// low/high value to controller ---------
      L     DB273.DBD   30; // !!! insert correct AnI !!!
      T     DB276.DBD  218;

      L     DB273.DBD   34; // !!! insert correct AnI !!!
      T     DB276.DBD  222;

NETWORK
TITLE =Sequence organisation

      CLR   ;
      =     M    122.2;

// SFM supply ----------------------------------------------------------------

// analog value to SFM spare -----------------------
      L     DB273.DBD  146;
      T     DB171.DBD 1122; // !!! insert correct SFM !!!

// analog value to SFM spare -----------------------
      L     DB273.DBD  266;
      T     DB171.DBD 1122; // !!! insert correct SFM !!!

// analog value to SFM spare -----------------------
      L     DB273.DBD  386;
      T     DB171.DBD 1122; // !!! insert correct SFM !!!

// sequencer ----------------------------------------------------------------
      A     DB173.DBX   43.1;
      S     DB173.DBX   97.3;

//      CALL  "SeO"          Called in Unit
//       UnitNo:=#UnitNo

NETWORK
TITLE =Auto / Manual

      SET   ;
      AN    M    122.2;
      JC    MODE;
      AN    M    120.1;


// assign PID mode
      S     DB276.DBX  201.4;
      S     DB276.DBX  201.5;


MODE: SET   ;

END_FUNCTION_BLOCK

FUNCTION_BLOCK FB 560
TITLE =
AUTHOR : RR
FAMILY : BOTEC_F1
NAME : OrLiMngA
VERSION : 1.0


VAR_TEMP
  RetVal : WORD ;	//return value
  ValDW : DWORD ;
  ValOK : BOOL ;
  SetValue : DWORD ;
END_VAR
BEGIN
NETWORK
TITLE =Send-/Receive manager telegramtype 1


// Send manager telegramtype 1
      CALL FC   571 (
           RET_VAL                  := #RetVal);

      JBI   OKS1; // Jump, if all OK
// Error evaluation
      L     #RetVal; // Return value
      L     DB33.DBD   84; // Error number from answer
OKS1: NOP   0;

// Receive manager telegramtype 1
      CALL FC   572 (
           RET_VAL                  := #RetVal);

      JBI   OKR1; // Jump, if all OK
// Error evaluation
      L     #RetVal; // Return value
      L     DB33.DBD   84; // Error number from answer
OKR1: NOP   0;


NETWORK
TITLE =Order management

// Telegramtype 1

      CALL FC   560 (
           OrLiDB                   := DB   561,
           RET_VAL                  := #RetVal);

// Telegramtype 2

      CALL FC   560 (
           OrLiDB                   := DB   562,
           RET_VAL                  := #RetVal);

// Telegramtype 3

      CALL FC   560 (
           OrLiDB                   := DB   563,
           RET_VAL                  := #RetVal);

// Telegramtype 4

      CALL FC   560 (
           OrLiDB                   := DB   564,
           RET_VAL                  := #RetVal);

// Telegramtype 5

      CALL FC   560 (
           OrLiDB                   := DB   565,
           RET_VAL                  := #RetVal);


NETWORK
TITLE =Buffer diagnosis

      UC    FB   575;


END_FUNCTION_BLOCK

FUNCTION_BLOCK FB 581
TITLE =
AUTHOR : RR
FAMILY : BOTEC_F1
NAME : CrCA
VERSION : 2.1


VAR_TEMP
  RemotePLCNo : INT ;	//remote PLC number
  RetVal : WORD ;	//return value
END_VAR
BEGIN
NETWORK
TITLE =coupling active bits initialize

      AN    M    101.4;
      JC    NCRC;
      R     DB580.DBX   23.4; // initialize active bits (reset)
      R     DB580.DBX   11.4;
      R     DB580.DBX   47.4;
      R     DB580.DBX   35.4;
      R     DB580.DBX   71.4;
      R     DB580.DBX   59.4;
      R     DB580.DBX   95.4;
      R     DB580.DBX   83.4;
      R     DB580.DBX  119.4;
      R     DB580.DBX  107.4;
      R     DB580.DBX  143.4;
      R     DB580.DBX  131.4;
      R     DB580.DBX  167.4;
      R     DB580.DBX  155.4;
      R     DB580.DBX  191.4;
      R     DB580.DBX  179.4;

NCRC: SET   ;
NETWORK
TITLE =read/write data from/to remote PLC

      NOP   0;

// PLC01
      CALL FB   580 , DB   581 (
           RemotePLCNo              := #RemotePLCNo,
           RetVal                   := #RetVal);

// PLC02
      CALL FB   580 , DB   582 (
           RemotePLCNo              := #RemotePLCNo,
           RetVal                   := #RetVal);

// PLC03
      CALL FB   580 , DB   583 (
           RemotePLCNo              := #RemotePLCNo,
           RetVal                   := #RetVal);

// PLC04
      CALL FB   580 , DB   584 (
           RemotePLCNo              := #RemotePLCNo,
           RetVal                   := #RetVal);

// PLC05
//      CALL  "CCL" , "CCLP05D"
//       RemotePLCNo:=#RemotePLCNo
//       RetVal     :=#RetVal

// PLC06
//      CALL  "CCL" , "CCLP06D"
//       RemotePLCNo:=#RemotePLCNo
//       RetVal     :=#RetVal

// PLC07
//      CALL  "CCL" , "CCLP07D"
//       RemotePLCNo:=#RemotePLCNo
//       RetVal     :=#RetVal

// PLC08
//      CALL  "CCL" , "CCLP08D"
//       RemotePLCNo:=#RemotePLCNo
//       RetVal     :=#RetVal

END_FUNCTION_BLOCK

FUNCTION_BLOCK FB 1000
TITLE =
FAMILY : BOTEC
NAME : UniA
VERSION : 2.0


VAR_TEMP
  UnitNo : INT ;	//unit number
END_VAR
BEGIN
NETWORK
TITLE =general

      L     DB1000.DBW    0;
      T     #UnitNo;

NETWORK
TITLE =analog input's

//      CALL  "AnI"
//       UnitNo:=#UnitNo
//       AnIRec:="U00AnID".AnI1
//       ValPer:=PEW1024

NETWORK
TITLE =PID controller assignment

//      CALL  "PID"
//       UnitNo:=#UnitNo
//       PIDRec:="U00PIDD".PID1
//       SpExt :"U01SeqD".Seq.SFM[x].Sp
//       PVal  :="U00AnID".AnI1.Val
//       OPer  :=PAW1024


//      CALL  "VLT"
//       UnitNo :=#UnitNo
//       VLTRec :="U00VLTD".VLT1
//       BasePEW:=PEW2048
//       COn    :="U00ActD".Act1.Out
//       SpExt  :="U00PIDD".PID1.OVal

NETWORK
TITLE =special input's

//      CALL  "SI1"
//       UnitNo:=#UnitNo
//       SpIRec:="U00SpID".SpI1
//       SpIBit:=E256.0

NETWORK
TITLE =counter

//      CALL  "Cnt"
//       UnitNo:=#UnitNo
//       CntRec:="U00CntD".Cnt1
//       Imp   :="U00SpID".SpI1.Sig
NETWORK
TITLE =message
//
//
// reserved

NETWORK
TITLE =sequence organisation call

      SET   ;
// assignment counter values

//       CALL  "C2S"
//       UnitNo:=#UnitNo
//       CntRec:="U00CntD".Cnt1
//       Enable:="OrgS1"
//       SFMRec:="U00SeqD".Seq.SFM[x]

// assignment analog values

//      L     "U00AnID".AnI1.Val
//      T     "U00SeqD".Seq.SFM[x].Val

      CALL FC    40 (
           UnitNo                   := #UnitNo);

NETWORK
TITLE =mode assignment actuators + PID-controllers

      AN    M    122.2;
      JC    MODE;

      AN    M    120.1;
//      =     "U00ActD".Act1.Auto


MODE: SET   ;
NETWORK
TITLE =actuator's


//      CALL  "Act"
//       UnitNo:=#UnitNo
//       ActRec:="U00ActD".Act1
//       Typ   :=1
//       FBa   :=E0.0
//       FBa2  :=E0.0
//       Out   :=A0.0

END_FUNCTION_BLOCK

FUNCTION_BLOCK FB 1010
TITLE =U001: Wassertank 01
FAMILY : BOTEC_F1
NAME : U001A
VERSION : 2.1


VAR_TEMP
  EStopOK : BOOL ;	//auxiliary flag
  CIP : BOOL ;	//CIP Program Selected
  xTmp : BOOL ;	//Temporary Bool(free for general use)
  DummyBool : BOOL ;	//Temporary Bool(free for general use)
  UnitNo : INT ;	//unit number
  UnitFB : INT ;	//unit expansion FB number
  rTmp : REAL ;	//Temporary REAL (free for general use)
  iTmp : INT ;	//Temporary INT (free for general use)
  DummyInt : INT ;	//Temporary INT (free for general use)
  dTmp : DINT ;	//Temporary DINT (free for general use)
END_VAR
BEGIN
NETWORK
TITLE =general

      CLR   ;
      =     #xTmp;
      =     #EStopOK;

      L     DB1010.DBW    0;
      T     #UnitNo;
      L     DB1010.DBW    2;
      T     #UnitFB;

NETWORK
TITLE =analog inputs

      NOP   0;
// LI_T1 AnI 001 Inhalt Tank 1
      CALL FC    24 (
           UnitNo                   := #UnitNo,
           AnIRec                   := DB2013.LI_T1,
           ValPer                   := DB302.DBW   64);

NETWORK
TITLE =Universal value

      NOP   0;
// unv001 UnV 001 Process Status
      CALL FC    27 (
           UnitNo                   := #UnitNo,
           UnVRec                   := DB2015.unv001,
           ValExt                   := DB2015.DBD  234);

// unv002 UnV 002 Universal Value 02
      CALL FC    27 (
           UnitNo                   := #UnitNo,
           UnVRec                   := DB2015.unv002,
           ValExt                   := DB2015.DBD  362);

// unv003 UnV 003 Universal Value 03
      CALL FC    27 (
           UnitNo                   := #UnitNo,
           UnVRec                   := DB2015.unv003,
           ValExt                   := DB2015.DBD  490);

NETWORK
TITLE =special inputs

      NOP   0;
// LS_LLL_T1 SpI 001
      CALL FC    14 (
           UnitNo                   := #UnitNo,
           SpIRec                   := DB2011.LS_LLL_T1,
           SpIBit                   := I     70.0);

// LS_HL_T1 SpI 002
      CALL FC    14 (
           UnitNo                   := #UnitNo,
           SpIRec                   := DB2011.LS_HL_T1,
           SpIBit                   := I     69.5);

// RM_NI_T1_VV SpI 004 Vacuumventil Tank 1
      CALL FC    14 (
           UnitNo                   := #UnitNo,
           SpIRec                   := DB2011.RM_NI_T1_VV,
           SpIBit                   := I    186.5);

// LS_LL_T1 SpI 005 (als Leermeldung ausgelegt)
      CALL FC    14 (
           UnitNo                   := #UnitNo,
           SpIRec                   := DB2011.LS_LL_T1,
           SpIBit                   := I     69.6);

// RM_NI_T1_K4_AUF SpI 006 Klappe vor Filter Tank 1
      CALL FC    14 (
           UnitNo                   := #UnitNo,
           SpIRec                   := DB2011.RM_NI_T1_K4_AUF,
           SpIBit                   := I    186.3);

// RM_NI_T1_K4_ZU SpI 007 Klappe vor Filter Tank 1
      CALL FC    14 (
           UnitNo                   := #UnitNo,
           SpIRec                   := DB2011.RM_NI_T1_K4_ZU,
           SpIBit                   := I    186.4);

// RM_NI_T1_K2 SpI 008 Handklappe Tank 1
      CALL FC    14 (
           UnitNo                   := #UnitNo,
           SpIRec                   := DB2011.RM_NI_T1_K2,
           SpIBit                   := I     71.1);

// RM_NI_T1_K3 SpI 010 Handklappe Tank 1
      CALL FC    14 (
           UnitNo                   := #UnitNo,
           SpIRec                   := DB2011.RM_NI_T1_K3,
           SpIBit                   := I     71.2);

// LABOR_FREIG_T1 SpI 011 SCHLUESSELSCHALTER LABOR
      CALL FC    14 (
           UnitNo                   := #UnitNo,
           SpIRec                   := DB2011.LABOR_FREIG_T1,
           SpIBit                   := I    258.0);

NETWORK
TITLE =messages

      NOP   0;
// msg001 Msg 001 Message 01
      CALL FC    16 (
           UnitNo                   := #UnitNo,
           MsgRec                   := DB2017.msg001,
           MsgBit                   := DB2017.DBX   82.7);

// msg002 Msg 002 Message 02
      CALL FC    16 (
           UnitNo                   := #UnitNo,
           MsgRec                   := DB2017.msg002,
           MsgBit                   := DB2017.DBX  142.7);

NETWORK
TITLE =unit supply

      UC    FB [#UnitFB];

NETWORK
TITLE =T1_A10
// Act 005
// Box           : Ventilinsel 2
// Input address : I317.0
// Output address: Q317.0
      CALL FC    70 (
           UnitNo                   := #UnitNo,
           ActRec                   := DB2010.T1_A10,
           Typ                      := 1,
           FBa                      := #xTmp,
           FBa2                     := I    317.0,
           Out                      := Q    317.0);

NETWORK
TITLE =T1_A9
// Act 006
// Box           : Ventilinsel 2
// Input address : I319.0
// Output address: Q319.0
      CALL FC    70 (
           UnitNo                   := #UnitNo,
           ActRec                   := DB2010.T1_A9,
           Typ                      := 1,
           FBa                      := #xTmp,
           FBa2                     := I    319.0,
           Out                      := Q    319.0);

NETWORK
TITLE =T1_A12
// Act 007
// Box           : Ventilinsel 2
// Input address : I321.0
// Output address: Q321.0
      CALL FC    70 (
           UnitNo                   := #UnitNo,
           ActRec                   := DB2010.T1_A12,
           Typ                      := 1,
           FBa                      := #xTmp,
           FBa2                     := I    321.0,
           Out                      := Q    321.0);

NETWORK
TITLE =T1_A7
// Act 008
// Box           : Ventilinsel 2
// Input address : I323.0
// Output address: Q323.0
      CALL FC    70 (
           UnitNo                   := #UnitNo,
           ActRec                   := DB2010.T1_A7,
           Typ                      := 1,
           FBa                      := #xTmp,
           FBa2                     := I    323.0,
           Out                      := Q    323.0);

NETWORK
TITLE =T1_A8
// Act 009
// Box           : Ventilinsel 3
// Input address : I325.0
// Output address: Q325.0
      CALL FC    70 (
           UnitNo                   := #UnitNo,
           ActRec                   := DB2010.T1_A8,
           Typ                      := 1,
           FBa                      := #xTmp,
           FBa2                     := I    325.0,
           Out                      := Q    325.0);

NETWORK
TITLE =T1_A5
// Act 010
// Box           : Ventilinsel 3
// Input address : I327.0
// Output address: Q327.0
      CALL FC    70 (
           UnitNo                   := #UnitNo,
           ActRec                   := DB2010.T1_A5,
           Typ                      := 1,
           FBa                      := #xTmp,
           FBa2                     := I    327.0,
           Out                      := Q    327.0);

NETWORK
TITLE =T1_A11
// Act 011
// Box           : Ventilinsel 3
// Input address : I329.0
// Output address: Q329.0
      CALL FC    70 (
           UnitNo                   := #UnitNo,
           ActRec                   := DB2010.T1_A11,
           Typ                      := 1,
           FBa                      := #xTmp,
           FBa2                     := I    329.0,
           Out                      := Q    329.0);

NETWORK
TITLE =T1_A14
// Act 012
// Box           : Ventilinsel 4
// Input address : I331.0
// Output address: Q331.0
      CALL FC    70 (
           UnitNo                   := #UnitNo,
           ActRec                   := DB2010.T1_A14,
           Typ                      := 1,
           FBa                      := #xTmp,
           FBa2                     := I    331.0,
           Out                      := Q    331.0);

NETWORK
TITLE =T1_A15
// Act 013
// Box           : Ventilinsel 4
// Input address : I333.0
// Output address: Q333.0
      CALL FC    70 (
           UnitNo                   := #UnitNo,
           ActRec                   := DB2010.T1_A15,
           Typ                      := 0,
           FBa                      := #xTmp,
           FBa2                     := I    333.0,
           Out                      := Q    333.0);

NETWORK
TITLE =T1_RR1
// Act 014
// Box           : Ventilinsel 4
// Input address : I335.0
// Output address: Q335.0
      CALL FC    70 (
           UnitNo                   := #UnitNo,
           ActRec                   := DB2010.T1_RR1,
           Typ                      := 1,
           FBa                      := #xTmp,
           FBa2                     := I    335.0,
           Out                      := Q    335.0);

NETWORK
TITLE =RV1_T1  RV1_T1
// Act 015
// Box           : VS1-BB
// Input address : I296.0
// Output address: Q296.0
      CALL FC    70 (
           UnitNo                   := #UnitNo,
           ActRec                   := DB2010.RV1_T1,
           Typ                      := 1,
           FBa                      := #xTmp,
           FBa2                     := I    296.0,
           Out                      := Q    296.0);

NETWORK
TITLE =B6F_T1  B6F_T1
// Act 016
// Box           : VS1-BB
// Input address : I296.4
// Output address: Q296.4
      CALL FC    70 (
           UnitNo                   := #UnitNo,
           ActRec                   := DB2010.B6F_T1,
           Typ                      := 1,
           FBa                      := #xTmp,
           FBa2                     := I    296.4,
           Out                      := Q    296.4);

NETWORK
TITLE =H6F_T1  H6F_T1
// Act 017
// Box           : VS1-BB
// Input address : I296.3
// Output address: Q296.3
      CALL FC    70 (
           UnitNo                   := #UnitNo,
           ActRec                   := DB2010.H6F_T1,
           Typ                      := 1,
           FBa                      := #xTmp,
           FBa2                     := I    296.3,
           Out                      := Q    296.3);

NETWORK
TITLE =J6F_T1  J6F_T1
// Act 018
// Box           : VS1-BB
// Input address : I296.5
// Output address: Q296.5
      CALL FC    70 (
           UnitNo                   := #UnitNo,
           ActRec                   := DB2010.J6F_T1,
           Typ                      := 1,
           FBa                      := #xTmp,
           FBa2                     := I    296.5,
           Out                      := Q    296.5);

NETWORK
TITLE =L6F_T1  L6F_T1
// Act 019
// Box           : VS1-BB
// Input address : I296.6
// Output address: Q296.6
      CALL FC    70 (
           UnitNo                   := #UnitNo,
           ActRec                   := DB2010.L6F_T1,
           Typ                      := 1,
           FBa                      := #xTmp,
           FBa2                     := I    296.6,
           Out                      := Q    296.6);

NETWORK
TITLE =D6_T1  D6_T1
// Act 020
// Box           : VS1-BB
// Input address : I297.0
// Output address: Q297.0
      CALL FC    70 (
           UnitNo                   := #UnitNo,
           ActRec                   := DB2010.D6_T1,
           Typ                      := 1,
           FBa                      := #xTmp,
           FBa2                     := I    297.0,
           Out                      := Q    297.0);

NETWORK
TITLE =B6_T1  B6_T1
// Act 021
// Box           : VS1-BB
// Input address : I296.7
// Output address: Q296.7
      CALL FC    70 (
           UnitNo                   := #UnitNo,
           ActRec                   := DB2010.B6_T1,
           Typ                      := 1,
           FBa                      := #xTmp,
           FBa2                     := I    296.7,
           Out                      := Q    296.7);

NETWORK
TITLE =A_T1  A_T1
// Act 022
// Box           : VS1-BB
// Input address : I296.1
// Output address: Q296.1
      CALL FC    70 (
           UnitNo                   := #UnitNo,
           ActRec                   := DB2010.A_T1,
           Typ                      := 1,
           FBa                      := #xTmp,
           FBa2                     := I    296.1,
           Out                      := Q    296.1);

NETWORK
TITLE =B_T1  B_T1
// Act 023
// Box           : VS1-BB
// Input address : I296.2
// Output address: Q296.2
      CALL FC    70 (
           UnitNo                   := #UnitNo,
           ActRec                   := DB2010.B_T1,
           Typ                      := 1,
           FBa                      := #xTmp,
           FBa2                     := I    296.2,
           Out                      := Q    296.2);

NETWORK
TITLE =CF_T1
// Act 024
// Box           : Ventilinsel 1
// Input address : I16.1
// Output address: Q16.1
      CALL FC    70 (
           UnitNo                   := #UnitNo,
           ActRec                   := DB2010.CF_T1,
           Typ                      := 1,
           FBa                      := #xTmp,
           FBa2                     := I     16.1,
           Out                      := Q     16.1);

NETWORK
TITLE =RW5_T1  Ansteuerung Befüllventil
// Act 026
// Box           : Ventilinsel 1
// Input address : I16.0
// Output address: Q16.0
      CALL FC    70 (
           UnitNo                   := #UnitNo,
           ActRec                   := DB2010.RW5_T1,
           Typ                      := 1,
           FBa                      := #xTmp,
           FBa2                     := I     16.0,
           Out                      := Q     16.0);

NETWORK
TITLE =RW6_T1  RW6_T1
// Act 027
// Box           : VS1-BB
// Input address : I297.1
// Output address: Q297.1
      CALL FC    70 (
           UnitNo                   := #UnitNo,
           ActRec                   := DB2010.RW6_T1,
           Typ                      := 1,
           FBa                      := #xTmp,
           FBa2                     := I    297.1,
           Out                      := Q    297.1);

NETWORK
TITLE =VR_T1  VR_T1
// Act 029
// Box           : VS1-BB
// Output address: Q297.2
      CALL FC    70 (
           UnitNo                   := #UnitNo,
           ActRec                   := DB2010.VR_T1,
           Typ                      := 0,
           FBa                      := #xTmp,
           FBa2                     := #xTmp,
           Out                      := Q    297.2);

NETWORK
TITLE =T1_V3
// Act 030
// Box           : Ventilinsel 5
// Input address : I340.2
// Output address: Q340.2
//      CALL  "Act"
//       UnitNo:=#UnitNo
//       ActRec:="U001ActD".T1_V3
//       Typ   :=0
//       FBa   :=#xTmp
//       FBa2  :="T1_V3GSC"
//       Out   :="T1_V3O"

NETWORK
TITLE =ML_LABORFREIGABE_T1
// Act 031
// Box           : LT-CIP
// Output address: Q258.0
      CALL FC    70 (
           UnitNo                   := #UnitNo,
           ActRec                   := DB2010.ML_LABORFREIGABE_T1,
           Typ                      := 0,
           FBa                      := #xTmp,
           FBa2                     := #xTmp,
           Out                      := Q    258.0);

END_FUNCTION_BLOCK

FUNCTION_BLOCK FB 1011
TITLE =U001: Water Tank 1
FAMILY : BOTEC_F1
NAME : UniE
VERSION : 1.2


VAR_TEMP
  CIP : BOOL ;	//CIP active
  UNIM : BOOL ;	//Unit Not In Maintenance
  GenRel : BOOL ;	//general OK (emergency and maintenance OK)
  EStopOK : BOOL ;	//emergency OK
  UnitNo : INT ;	//unit number
  xTmp : BOOL ;	//Temporary Bool
  iTmp : INT ;	//Temporary INT
  rTmp : REAL ;	//Temporary REAL
  dTmp : DINT ;	//Temporary DINT (free for general use)
  RetValInt : INT ;	//return value
END_VAR
BEGIN
NETWORK
TITLE =General

      SET   ;
// Simulation ---------------------------------------------------------------
      A     DB1011.DBX 1357.7;
      CC    FB  1019; // "U001Sim"
      A     DB1011.DBX   17.3;
      =     DB1011.DBX 1357.7; //Help bit for simulation

// get unit number ----------------------------------------------------------
      L     DB1010.DBW    0;
      T     #UnitNo;

// communication ------------------------------------------------------------
      UC    FB  1015; // U001Com

NETWORK
TITLE =Sequence organisation

      CLR   ;
      =     M    122.2;

// CIP Counter
      CALL FC    29 (
           UnitNo                   := #UnitNo,
           Value                    := DB1015.DBD   54,
           Enable                   := TRUE,
           Down                     := FALSE,
           OriginDetect             := 0.000000e+000,
           MaxDiffPS                := 1.000000e+000,
           SFMRec                   := DB1011.Seq.SFM[15],
           ValueOld                 := DB1011.DBD 1418);

// sequencer ----------------------------------------------------------------
      A     DB1013.DBX   43.1;
      S     DB1013.DBX   97.3;

      CALL FC    40 (
           UnitNo                   := #UnitNo);

END_FUNCTION_BLOCK

FUNCTION_BLOCK FB 1020
TITLE =U002: Wassertank 02
FAMILY : BOTEC_F1
NAME : U002A
VERSION : 2.1


VAR_TEMP
  EStopOK : BOOL ;	//auxiliary flag
  CIP : BOOL ;	//CIP Program Selected
  xTmp : BOOL ;	//Temporary Bool(free for general use)
  DummyBool : BOOL ;	//Temporary Bool(free for general use)
  UnitNo : INT ;	//unit number
  UnitFB : INT ;	//unit expansion FB number
  rTmp : REAL ;	//Temporary REAL (free for general use)
  iTmp : INT ;	//Temporary INT (free for general use)
  DummyInt : INT ;	//Temporary INT (free for general use)
  dTmp : DINT ;	//Temporary DINT (free for general use)
END_VAR
BEGIN
NETWORK
TITLE =general

      CLR   ;
      =     #xTmp;
      =     #EStopOK;

      L     DB1020.DBW    0;
      T     #UnitNo;
      L     DB1020.DBW    2;
      T     #UnitFB;

NETWORK
TITLE =analog inputs

      NOP   0;
// LI_T2 AnI 001 Inhalt Tank 2
      CALL FC    24 (
           UnitNo                   := #UnitNo,
           AnIRec                   := DB2023.LI_T2,
           ValPer                   := DB302.DBW   66);

NETWORK
TITLE =Universal value

      NOP   0;
// unv001 UnV 001 Process Status
      CALL FC    27 (
           UnitNo                   := #UnitNo,
           UnVRec                   := DB2025.unv001,
           ValExt                   := DB2025.DBD  234);

// unv002 UnV 002 Universal Value 02
      CALL FC    27 (
           UnitNo                   := #UnitNo,
           UnVRec                   := DB2025.unv002,
           ValExt                   := DB2025.DBD  362);

// unv003 UnV 003 Universal Value 03
      CALL FC    27 (
           UnitNo                   := #UnitNo,
           UnVRec                   := DB2025.unv003,
           ValExt                   := DB2025.DBD  490);

NETWORK
TITLE =special inputs

      NOP   0;
// LS_LLL_T2 SpI 001
      CALL FC    14 (
           UnitNo                   := #UnitNo,
           SpIRec                   := DB2021.LS_LLL_T2,
           SpIBit                   := I     71.7);

// LS_HL_T2 SpI 002
      CALL FC    14 (
           UnitNo                   := #UnitNo,
           SpIRec                   := DB2021.LS_HL_T2,
           SpIBit                   := I     69.7);

// LS_LL_T2 SpI 005
      CALL FC    14 (
           UnitNo                   := #UnitNo,
           SpIRec                   := DB2021.LS_LL_T2,
           SpIBit                   := I     70.1);

// RM_NI_T2_K2 SpI 008
      CALL FC    14 (
           UnitNo                   := #UnitNo,
           SpIRec                   := DB2021.RM_NI_T2_K2,
           SpIBit                   := I     61.6);

// RM_NI_T2_K3 SpI 010
      CALL FC    14 (
           UnitNo                   := #UnitNo,
           SpIRec                   := DB2021.RM_NI_T2_K3,
           SpIBit                   := I     61.7);

// LABOR_FREIG_T2 SpI 011 SCHLUESSELSCHALTER LABOR
      CALL FC    14 (
           UnitNo                   := #UnitNo,
           SpIRec                   := DB2021.LABOR_FREIG_T2,
           SpIBit                   := I    258.1);

NETWORK
TITLE =messages

      NOP   0;
// msg001 Msg 001 Message 01
      CALL FC    16 (
           UnitNo                   := #UnitNo,
           MsgRec                   := DB2027.msg001,
           MsgBit                   := DB2027.DBX   82.7);

// msg002 Msg 002 Message 02
      CALL FC    16 (
           UnitNo                   := #UnitNo,
           MsgRec                   := DB2027.msg002,
           MsgBit                   := DB2027.DBX  142.7);

NETWORK
TITLE =unit supply

      UC    FB [#UnitFB];

NETWORK
TITLE =T2_A10
// Act 005
// Box           : Ventilinsel 2
// Input address : I316.7
// Output address: Q316.7
      CALL FC    70 (
           UnitNo                   := #UnitNo,
           ActRec                   := DB2020.T2_A10,
           Typ                      := 1,
           FBa                      := #xTmp,
           FBa2                     := I    316.7,
           Out                      := Q    316.7);

NETWORK
TITLE =T2_A9
// Act 006
// Box           : Ventilinsel 2
// Input address : I318.7
// Output address: Q318.7
      CALL FC    70 (
           UnitNo                   := #UnitNo,
           ActRec                   := DB2020.T2_A9,
           Typ                      := 1,
           FBa                      := #xTmp,
           FBa2                     := I    318.7,
           Out                      := Q    318.7);

NETWORK
TITLE =T2_A12
// Act 007
// Box           : Ventilinsel 2
// Input address : I320.7
// Output address: Q320.7
      CALL FC    70 (
           UnitNo                   := #UnitNo,
           ActRec                   := DB2020.T2_A12,
           Typ                      := 1,
           FBa                      := #xTmp,
           FBa2                     := I    320.7,
           Out                      := Q    320.7);

NETWORK
TITLE =T2_A7
// Act 008
// Box           : Ventilinsel 2
// Input address : I322.7
// Output address: Q322.7
      CALL FC    70 (
           UnitNo                   := #UnitNo,
           ActRec                   := DB2020.T2_A7,
           Typ                      := 1,
           FBa                      := #xTmp,
           FBa2                     := I    322.7,
           Out                      := Q    322.7);

NETWORK
TITLE =T2_A8
// Act 009
// Box           : Ventilinsel 3
// Input address : I324.7
// Output address: Q324.7
      CALL FC    70 (
           UnitNo                   := #UnitNo,
           ActRec                   := DB2020.T2_A8,
           Typ                      := 1,
           FBa                      := #xTmp,
           FBa2                     := I    324.7,
           Out                      := Q    324.7);

NETWORK
TITLE =T2_A5
// Act 010
// Box           : Ventilinsel 3
// Input address : I326.7
// Output address: Q326.7
      CALL FC    70 (
           UnitNo                   := #UnitNo,
           ActRec                   := DB2020.T2_A5,
           Typ                      := 1,
           FBa                      := #xTmp,
           FBa2                     := I    326.7,
           Out                      := Q    326.7);

NETWORK
TITLE =T2_A11
// Act 011
// Box           : Ventilinsel 3
// Input address : I328.7
// Output address: Q328.7
      CALL FC    70 (
           UnitNo                   := #UnitNo,
           ActRec                   := DB2020.T2_A11,
           Typ                      := 1,
           FBa                      := #xTmp,
           FBa2                     := I    328.7,
           Out                      := Q    328.7);

NETWORK
TITLE =T2_A14
// Act 012
// Box           : Ventilinsel 4
// Input address : I330.7
// Output address: Q330.7
      CALL FC    70 (
           UnitNo                   := #UnitNo,
           ActRec                   := DB2020.T2_A14,
           Typ                      := 1,
           FBa                      := #xTmp,
           FBa2                     := I    330.7,
           Out                      := Q    330.7);

NETWORK
TITLE =T2_A15
// Act 013
// Box           : Ventilinsel 4
// Input address : I332.7
// Output address: Q332.7
      CALL FC    70 (
           UnitNo                   := #UnitNo,
           ActRec                   := DB2020.T2_A15,
           Typ                      := 0,
           FBa                      := #xTmp,
           FBa2                     := I    332.7,
           Out                      := Q    332.7);

NETWORK
TITLE =T2_RR1
// Act 014
// Box           : Ventilinsel 4
// Input address : I334.7
// Output address: Q334.7
      CALL FC    70 (
           UnitNo                   := #UnitNo,
           ActRec                   := DB2020.T2_RR1,
           Typ                      := 1,
           FBa                      := #xTmp,
           FBa2                     := I    334.7,
           Out                      := Q    334.7);

NETWORK
TITLE =RV1_T2  RV1_T2
// Act 015
// Box           : VS1-BB
// Input address : I297.3
// Output address: Q297.3
      CALL FC    70 (
           UnitNo                   := #UnitNo,
           ActRec                   := DB2020.RV1_T2,
           Typ                      := 1,
           FBa                      := #xTmp,
           FBa2                     := I    297.3,
           Out                      := Q    297.3);

NETWORK
TITLE =B6F_T2  B6F_T2
// Act 016
// Box           : VS1-BB
// Input address : I297.7
// Output address: Q297.7
      CALL FC    70 (
           UnitNo                   := #UnitNo,
           ActRec                   := DB2020.B6F_T2,
           Typ                      := 1,
           FBa                      := #xTmp,
           FBa2                     := I    297.7,
           Out                      := Q    297.7);

NETWORK
TITLE =H6F_T2  H6F_T2
// Act 017
// Box           : VS1-BB
// Input address : I297.6
// Output address: Q297.6
      CALL FC    70 (
           UnitNo                   := #UnitNo,
           ActRec                   := DB2020.H6F_T2,
           Typ                      := 1,
           FBa                      := #xTmp,
           FBa2                     := I    297.6,
           Out                      := Q    297.6);

NETWORK
TITLE =J6F_T2  J6F_T2
// Act 018
// Box           : VS1-BB
// Input address : I298.0
// Output address: Q298.0
      CALL FC    70 (
           UnitNo                   := #UnitNo,
           ActRec                   := DB2020.J6F_T2,
           Typ                      := 1,
           FBa                      := #xTmp,
           FBa2                     := I    298.0,
           Out                      := Q    298.0);

NETWORK
TITLE =L6F_T2  L6F_T2
// Act 019
// Box           : VS1-BB
// Input address : I298.1
// Output address: Q298.1
      CALL FC    70 (
           UnitNo                   := #UnitNo,
           ActRec                   := DB2020.L6F_T2,
           Typ                      := 1,
           FBa                      := #xTmp,
           FBa2                     := I    298.1,
           Out                      := Q    298.1);

NETWORK
TITLE =D6_T2  D6_T2
// Act 020
// Box           : VS1-BB
// Input address : I298.3
// Output address: Q298.3
      CALL FC    70 (
           UnitNo                   := #UnitNo,
           ActRec                   := DB2020.D6_T2,
           Typ                      := 1,
           FBa                      := #xTmp,
           FBa2                     := I    298.3,
           Out                      := Q    298.3);

NETWORK
TITLE =B6_T2  B6_T2
// Act 021
// Box           : VS1-BB
// Input address : I298.2
// Output address: Q298.2
      CALL FC    70 (
           UnitNo                   := #UnitNo,
           ActRec                   := DB2020.B6_T2,
           Typ                      := 1,
           FBa                      := #xTmp,
           FBa2                     := I    298.2,
           Out                      := Q    298.2);

NETWORK
TITLE =A_T2  A_T2
// Act 022
// Box           : VS1-BB
// Input address : I297.4
// Output address: Q297.4
      CALL FC    70 (
           UnitNo                   := #UnitNo,
           ActRec                   := DB2020.A_T2,
           Typ                      := 1,
           FBa                      := #xTmp,
           FBa2                     := I    297.4,
           Out                      := Q    297.4);

NETWORK
TITLE =B_T2  B_T2
// Act 023
// Box           : VS1-BB
// Input address : I297.5
// Output address: Q297.5
      CALL FC    70 (
           UnitNo                   := #UnitNo,
           ActRec                   := DB2020.B_T2,
           Typ                      := 1,
           FBa                      := #xTmp,
           FBa2                     := I    297.5,
           Out                      := Q    297.5);

NETWORK
TITLE =CF_T2
// Act 024
// Box           : Ventilinsel 1
// Input address : I16.2
// Output address: Q16.2
      CALL FC    70 (
           UnitNo                   := #UnitNo,
           ActRec                   := DB2020.CF_T2,
           Typ                      := 1,
           FBa                      := #xTmp,
           FBa2                     := I     16.2,
           Out                      := Q     16.2);

NETWORK
TITLE =VR_T2  VR_T2
// Act 029
// Box           : VS1-BB
// Output address: Q298.4
      CALL FC    70 (
           UnitNo                   := #UnitNo,
           ActRec                   := DB2020.VR_T2,
           Typ                      := 0,
           FBa                      := #xTmp,
           FBa2                     := #xTmp,
           Out                      := Q    298.4);

NETWORK
TITLE =ML_LABORFREIGABE_T2
// Act 031
// Box           : LT-CIP
// Output address: Q258.1
      CALL FC    70 (
           UnitNo                   := #UnitNo,
           ActRec                   := DB2020.ML_LABORFREIGABE_T2,
           Typ                      := 0,
           FBa                      := #xTmp,
           FBa2                     := #xTmp,
           Out                      := Q    258.1);

END_FUNCTION_BLOCK

FUNCTION_BLOCK FB 1021
TITLE =U002: Water Tank 2
FAMILY : BOTEC_F1
NAME : UniE
VERSION : 1.2


VAR_TEMP
  CIP : BOOL ;	//CIP active
  UNIM : BOOL ;	//Unit Not In Maintenance
  GenRel : BOOL ;	//general OK (emergency and maintenance OK)
  EStopOK : BOOL ;	//emergency OK
  UnitNo : INT ;	//unit number
  xTmp : BOOL ;	//Temporary Bool
  iTmp : INT ;	//Temporary INT
  rTmp : REAL ;	//Temporary REAL
  dTmp : DINT ;	//Temporary DINT (free for general use)
  RetValInt : INT ;	//return value
END_VAR
BEGIN
NETWORK
TITLE =General

      SET   ;
// Simulation ---------------------------------------------------------------
      A     DB1021.DBX 1357.7;
      CC    FB  1029; // "WT02Sim"
      A     DB1021.DBX   17.3;
      =     DB1021.DBX 1357.7; //Help bit for simulation

// get unit number ----------------------------------------------------------
      L     DB1020.DBW    0;
      T     #UnitNo;


// communication ------------------------------------------------------------
      UC    FB  1025; // WT02Com

NETWORK
TITLE =Sequence organisation

      CLR   ;
      =     M    122.2;

// CIP Counter
      CALL FC    29 (
           UnitNo                   := #UnitNo,
           Value                    := DB1025.DBD   54,
           Enable                   := TRUE,
           Down                     := FALSE,
           OriginDetect             := 0.000000e+000,
           MaxDiffPS                := 1.000000e+000,
           SFMRec                   := DB1021.Seq.SFM[15],
           ValueOld                 := DB1021.DBD 1418);

// sequencer ----------------------------------------------------------------
      A     DB1023.DBX   43.1;
      S     DB1023.DBX   97.3;

      CALL FC    40 (
           UnitNo                   := #UnitNo);

END_FUNCTION_BLOCK

FUNCTION_BLOCK FB 1030
TITLE =U003: Wassertank 03
FAMILY : BOTEC_F1
NAME : U003A
VERSION : 2.1


VAR_TEMP
  EStopOK : BOOL ;	//auxiliary flag
  CIP : BOOL ;	//CIP Program Selected
  xTmp : BOOL ;	//Temporary Bool(free for general use)
  DummyBool : BOOL ;	//Temporary Bool(free for general use)
  UnitNo : INT ;	//unit number
  UnitFB : INT ;	//unit expansion FB number
  rTmp : REAL ;	//Temporary REAL (free for general use)
  iTmp : INT ;	//Temporary INT (free for general use)
  DummyInt : INT ;	//Temporary INT (free for general use)
  dTmp : DINT ;	//Temporary DINT (free for general use)
END_VAR
BEGIN
NETWORK
TITLE =general

      CLR   ;
      =     #xTmp;
      =     #EStopOK;

      L     DB1030.DBW    0;
      T     #UnitNo;
      L     DB1030.DBW    2;
      T     #UnitFB;

NETWORK
TITLE =analog inputs

      NOP   0;
// LI_T3 AnI 001 Inhalt Tank 3
      CALL FC    24 (
           UnitNo                   := #UnitNo,
           AnIRec                   := DB2033.LI_T3,
           ValPer                   := DB302.DBW   68);

NETWORK
TITLE =Universal value

      NOP   0;
// unv001 UnV 001 Process Status
      CALL FC    27 (
           UnitNo                   := #UnitNo,
           UnVRec                   := DB2035.unv001,
           ValExt                   := DB2035.DBD  234);

// unv002 UnV 002 Universal Value 02
      CALL FC    27 (
           UnitNo                   := #UnitNo,
           UnVRec                   := DB2035.unv002,
           ValExt                   := DB2035.DBD  362);

// unv003 UnV 003 Universal Value 03
      CALL FC    27 (
           UnitNo                   := #UnitNo,
           UnVRec                   := DB2035.unv003,
           ValExt                   := DB2035.DBD  490);

NETWORK
TITLE =special inputs

      NOP   0;
// LS_LLL_T3 SpI 001
      CALL FC    14 (
           UnitNo                   := #UnitNo,
           SpIRec                   := DB2031.LS_LLL_T3,
           SpIBit                   := I     60.1);

// LS_HL_T3 SpI 002
      CALL FC    14 (
           UnitNo                   := #UnitNo,
           SpIRec                   := DB2031.LS_HL_T3,
           SpIBit                   := I     70.2);

// LS_LL_T3 SpI 005
      CALL FC    14 (
           UnitNo                   := #UnitNo,
           SpIRec                   := DB2031.LS_LL_T3,
           SpIBit                   := I     60.0);

// RM_NI_T3_K2 SpI 008
      CALL FC    14 (
           UnitNo                   := #UnitNo,
           SpIRec                   := DB2031.RM_NI_T3_K2,
           SpIBit                   := I     60.6);

// RM_NI_T3_K3 SpI 010
      CALL FC    14 (
           UnitNo                   := #UnitNo,
           SpIRec                   := DB2031.RM_NI_T3_K3,
           SpIBit                   := I     69.0);

// LABOR_FREIG_T3 SpI 011 SCHLUESSELSCHALTER LABOR
      CALL FC    14 (
           UnitNo                   := #UnitNo,
           SpIRec                   := DB2031.LABOR_FREIG_T3,
           SpIBit                   := I    258.2);

NETWORK
TITLE =messages

      NOP   0;
// msg001 Msg 001 Message 01
      CALL FC    16 (
           UnitNo                   := #UnitNo,
           MsgRec                   := DB2037.msg001,
           MsgBit                   := DB2037.DBX   82.7);

// msg002 Msg 002 Message 02
      CALL FC    16 (
           UnitNo                   := #UnitNo,
           MsgRec                   := DB2037.msg002,
           MsgBit                   := DB2037.DBX  142.7);

NETWORK
TITLE =unit supply

      UC    FB [#UnitFB];

NETWORK
TITLE =T3_A10
// Act 005
// Box           : Ventilinsel 2
// Input address : I316.6
// Output address: Q316.6
      CALL FC    70 (
           UnitNo                   := #UnitNo,
           ActRec                   := DB2030.T3_A10,
           Typ                      := 1,
           FBa                      := #xTmp,
           FBa2                     := I    316.6,
           Out                      := Q    316.6);

NETWORK
TITLE =T3_A9
// Act 006
// Box           : Ventilinsel 2
// Input address : I318.6
// Output address: Q318.6
      CALL FC    70 (
           UnitNo                   := #UnitNo,
           ActRec                   := DB2030.T3_A9,
           Typ                      := 1,
           FBa                      := #xTmp,
           FBa2                     := I    318.6,
           Out                      := Q    318.6);

NETWORK
TITLE =T3_A12
// Act 007
// Box           : Ventilinsel 2
// Input address : I320.6
// Output address: Q320.6
      CALL FC    70 (
           UnitNo                   := #UnitNo,
           ActRec                   := DB2030.T3_A12,
           Typ                      := 1,
           FBa                      := #xTmp,
           FBa2                     := I    320.6,
           Out                      := Q    320.6);

NETWORK
TITLE =T3_A7
// Act 008
// Box           : Ventilinsel 2
// Input address : I322.6
// Output address: Q322.6
      CALL FC    70 (
           UnitNo                   := #UnitNo,
           ActRec                   := DB2030.T3_A7,
           Typ                      := 1,
           FBa                      := #xTmp,
           FBa2                     := I    322.6,
           Out                      := Q    322.6);

NETWORK
TITLE =T3_A8
// Act 009
// Box           : Ventilinsel 3
// Input address : I324.6
// Output address: Q324.6
      CALL FC    70 (
           UnitNo                   := #UnitNo,
           ActRec                   := DB2030.T3_A8,
           Typ                      := 1,
           FBa                      := #xTmp,
           FBa2                     := I    324.6,
           Out                      := Q    324.6);

NETWORK
TITLE =T3_A5
// Act 010
// Box           : Ventilinsel 3
// Input address : I326.6
// Output address: Q326.6
      CALL FC    70 (
           UnitNo                   := #UnitNo,
           ActRec                   := DB2030.T3_A5,
           Typ                      := 1,
           FBa                      := #xTmp,
           FBa2                     := I    326.6,
           Out                      := Q    326.6);

NETWORK
TITLE =T3_A11
// Act 011
// Box           : Ventilinsel 3
// Input address : I328.6
// Output address: Q328.6
      CALL FC    70 (
           UnitNo                   := #UnitNo,
           ActRec                   := DB2030.T3_A11,
           Typ                      := 1,
           FBa                      := #xTmp,
           FBa2                     := I    328.6,
           Out                      := Q    328.6);

NETWORK
TITLE =T3_A14
// Act 012
// Box           : Ventilinsel 4
// Input address : I330.6
// Output address: Q330.6
      CALL FC    70 (
           UnitNo                   := #UnitNo,
           ActRec                   := DB2030.T3_A14,
           Typ                      := 1,
           FBa                      := #xTmp,
           FBa2                     := I    330.6,
           Out                      := Q    330.6);

NETWORK
TITLE =T3_A15
// Act 013
// Box           : Ventilinsel 4
// Input address : I332.6
// Output address: Q332.6
      CALL FC    70 (
           UnitNo                   := #UnitNo,
           ActRec                   := DB2030.T3_A15,
           Typ                      := 0,
           FBa                      := #xTmp,
           FBa2                     := I    332.6,
           Out                      := Q    332.6);

NETWORK
TITLE =T3_RR1
// Act 014
// Box           : Ventilinsel 4
// Input address : I334.6
// Output address: Q334.6
      CALL FC    70 (
           UnitNo                   := #UnitNo,
           ActRec                   := DB2030.T3_RR1,
           Typ                      := 1,
           FBa                      := #xTmp,
           FBa2                     := I    334.6,
           Out                      := Q    334.6);

NETWORK
TITLE =RV1_T3  RV1_T3 Ventil CIP Vorlauf Tank 3
// Act 015
// Box           : VS1-BB
// Input address : I298.5
// Output address: Q298.5
      CALL FC    70 (
           UnitNo                   := #UnitNo,
           ActRec                   := DB2030.RV1_T3,
           Typ                      := 1,
           FBa                      := #xTmp,
           FBa2                     := I    298.5,
           Out                      := Q    298.5);

NETWORK
TITLE =B6F_T3  B6F_T3
// Act 016
// Box           : VS1-BB
// Input address : I299.1
// Output address: Q299.1
      CALL FC    70 (
           UnitNo                   := #UnitNo,
           ActRec                   := DB2030.B6F_T3,
           Typ                      := 1,
           FBa                      := #xTmp,
           FBa2                     := I    299.1,
           Out                      := Q    299.1);

NETWORK
TITLE =H6F_T3  H6F_T3
// Act 017
// Box           : VS1-BB
// Input address : I299.0
// Output address: Q299.0
      CALL FC    70 (
           UnitNo                   := #UnitNo,
           ActRec                   := DB2030.H6F_T3,
           Typ                      := 1,
           FBa                      := #xTmp,
           FBa2                     := I    299.0,
           Out                      := Q    299.0);

NETWORK
TITLE =J6F_T3  J6F_T3
// Act 018
// Box           : VS1-BB
// Input address : I299.2
// Output address: Q299.2
      CALL FC    70 (
           UnitNo                   := #UnitNo,
           ActRec                   := DB2030.J6F_T3,
           Typ                      := 1,
           FBa                      := #xTmp,
           FBa2                     := I    299.2,
           Out                      := Q    299.2);

NETWORK
TITLE =L6F_T3  L6F_T3
// Act 019
// Box           : VS1-BB
// Input address : I299.3
// Output address: Q299.3
      CALL FC    70 (
           UnitNo                   := #UnitNo,
           ActRec                   := DB2030.L6F_T3,
           Typ                      := 1,
           FBa                      := #xTmp,
           FBa2                     := I    299.3,
           Out                      := Q    299.3);

NETWORK
TITLE =D6_T3  D6_T3
// Act 020
// Box           : VS1-BB
// Input address : I299.5
// Output address: Q299.5
      CALL FC    70 (
           UnitNo                   := #UnitNo,
           ActRec                   := DB2030.D6_T3,
           Typ                      := 1,
           FBa                      := #xTmp,
           FBa2                     := I    299.5,
           Out                      := Q    299.5);

NETWORK
TITLE =B6_T3  B6_T3
// Act 021
// Box           : VS1-BB
// Input address : I299.4
// Output address: Q299.4
      CALL FC    70 (
           UnitNo                   := #UnitNo,
           ActRec                   := DB2030.B6_T3,
           Typ                      := 1,
           FBa                      := #xTmp,
           FBa2                     := I    299.4,
           Out                      := Q    299.4);

NETWORK
TITLE =A_T3  A_T3
// Act 022
// Box           : VS1-BB
// Input address : I298.6
// Output address: Q298.6
      CALL FC    70 (
           UnitNo                   := #UnitNo,
           ActRec                   := DB2030.A_T3,
           Typ                      := 1,
           FBa                      := #xTmp,
           FBa2                     := I    298.6,
           Out                      := Q    298.6);

NETWORK
TITLE =B_T3  B_T3
// Act 023
// Box           : VS1-BB
// Input address : I298.7
// Output address: Q298.7
      CALL FC    70 (
           UnitNo                   := #UnitNo,
           ActRec                   := DB2030.B_T3,
           Typ                      := 1,
           FBa                      := #xTmp,
           FBa2                     := I    298.7,
           Out                      := Q    298.7);

NETWORK
TITLE =CF_T3
// Act 024
// Box           : Ventilinsel 1
// Input address : I16.3
// Output address: Q16.3
      CALL FC    70 (
           UnitNo                   := #UnitNo,
           ActRec                   := DB2030.CF_T3,
           Typ                      := 1,
           FBa                      := #xTmp,
           FBa2                     := I     16.3,
           Out                      := Q     16.3);

NETWORK
TITLE =VR_T3  VR_T3
// Act 029
// Box           : VS1-BB
// Output address: Q299.6
      CALL FC    70 (
           UnitNo                   := #UnitNo,
           ActRec                   := DB2030.VR_T3,
           Typ                      := 0,
           FBa                      := #xTmp,
           FBa2                     := #xTmp,
           Out                      := Q    299.6);

NETWORK
TITLE =ML_LABORFREIGABE_T3
// Act 031
// Box           : LT-CIP
// Output address: Q258.2
      CALL FC    70 (
           UnitNo                   := #UnitNo,
           ActRec                   := DB2030.ML_LABORFREIGABE_T3,
           Typ                      := 0,
           FBa                      := #xTmp,
           FBa2                     := #xTmp,
           Out                      := Q    258.2);

END_FUNCTION_BLOCK

FUNCTION_BLOCK FB 1031
TITLE =U003: Water Tank 3
FAMILY : BOTEC_F1
NAME : UniE
VERSION : 1.2


VAR_TEMP
  CIP : BOOL ;	//CIP active
  UNIM : BOOL ;	//Unit Not In Maintenance
  GenRel : BOOL ;	//general OK (emergency and maintenance OK)
  EStopOK : BOOL ;	//emergency OK
  UnitNo : INT ;	//unit number
  xTmp : BOOL ;	//Temporary Bool
  iTmp : INT ;	//Temporary INT
  rTmp : REAL ;	//Temporary REAL
  dTmp : DINT ;	//Temporary DINT (free for general use)
  RetValInt : INT ;	//return value
END_VAR
BEGIN
NETWORK
TITLE =General

      SET   ;
// Simulation ---------------------------------------------------------------
      A     DB1031.DBX 1357.7;
      CC    FB  1039; // "WT03Sim"
      A     DB1031.DBX   17.3;
      =     DB1031.DBX 1357.7; //Help bit for simulation

// get unit number ----------------------------------------------------------
      L     DB1030.DBW    0;
      T     #UnitNo;

// communication ------------------------------------------------------------
      UC    FB  1035; // WT03Com

NETWORK
TITLE =Sequence organisation

      CLR   ;
      =     M    122.2;

// CIP Counter
      CALL FC    29 (
           UnitNo                   := #UnitNo,
           Value                    := DB1035.DBD   54,
           Enable                   := TRUE,
           Down                     := FALSE,
           OriginDetect             := 0.000000e+000,
           MaxDiffPS                := 1.000000e+000,
           SFMRec                   := DB1031.Seq.SFM[15],
           ValueOld                 := DB1031.DBD 1418);

// sequencer ----------------------------------------------------------------
      A     DB1033.DBX   43.1;
      S     DB1033.DBX   97.3;

      CALL FC    40 (
           UnitNo                   := #UnitNo);

END_FUNCTION_BLOCK

FUNCTION_BLOCK FB 1040
TITLE =U004: Wassertank 04
FAMILY : BOTEC_F1
NAME : U004A
VERSION : 2.1


VAR_TEMP
  EStopOK : BOOL ;	//auxiliary flag
  CIP : BOOL ;	//CIP Program Selected
  xTmp : BOOL ;	//Temporary Bool(free for general use)
  DummyBool : BOOL ;	//Temporary Bool(free for general use)
  UnitNo : INT ;	//unit number
  UnitFB : INT ;	//unit expansion FB number
  rTmp : REAL ;	//Temporary REAL (free for general use)
  iTmp : INT ;	//Temporary INT (free for general use)
  DummyInt : INT ;	//Temporary INT (free for general use)
  dTmp : DINT ;	//Temporary DINT (free for general use)
END_VAR
BEGIN
NETWORK
TITLE =general

      CLR   ;
      =     #xTmp;
      =     #EStopOK;

      L     DB1040.DBW    0;
      T     #UnitNo;
      L     DB1040.DBW    2;
      T     #UnitFB;

NETWORK
TITLE =analog inputs

      NOP   0;
// LI_T4 AnI 001 Inhalt Tank 4
      CALL FC    24 (
           UnitNo                   := #UnitNo,
           AnIRec                   := DB2043.LI_T4,
           ValPer                   := DB302.DBW   70);

NETWORK
TITLE =Universal value

      NOP   0;
// unv001 UnV 001 Process Status
      CALL FC    27 (
           UnitNo                   := #UnitNo,
           UnVRec                   := DB2045.unv001,
           ValExt                   := DB2045.DBD  234);

// unv002 UnV 002 Universal Value 02
      CALL FC    27 (
           UnitNo                   := #UnitNo,
           UnVRec                   := DB2045.unv002,
           ValExt                   := DB2045.DBD  362);

// unv003 UnV 003 Universal Value 03
      CALL FC    27 (
           UnitNo                   := #UnitNo,
           UnVRec                   := DB2045.unv003,
           ValExt                   := DB2045.DBD  490);

NETWORK
TITLE =special inputs

      NOP   0;
// LS_LLL_T4 SpI 001
      CALL FC    14 (
           UnitNo                   := #UnitNo,
           SpIRec                   := DB2041.LS_LLL_T4,
           SpIBit                   := I     67.4);

// LS_HL_T4 SpI 002
      CALL FC    14 (
           UnitNo                   := #UnitNo,
           SpIRec                   := DB2041.LS_HL_T4,
           SpIBit                   := I     67.2);

// LS_LL_T4 SpI 005
      CALL FC    14 (
           UnitNo                   := #UnitNo,
           SpIRec                   := DB2041.LS_LL_T4,
           SpIBit                   := I     67.3);

// RM_NI_T4_K2 SpI 008
      CALL FC    14 (
           UnitNo                   := #UnitNo,
           SpIRec                   := DB2041.RM_NI_T4_K2,
           SpIBit                   := I     60.7);

// RM_NI_T4_K3 SpI 010
      CALL FC    14 (
           UnitNo                   := #UnitNo,
           SpIRec                   := DB2041.RM_NI_T4_K3,
           SpIBit                   := I     69.1);

// LABOR_FREIG_T4 SpI 011 SCHLUESSELSCHALTER LABOR
      CALL FC    14 (
           UnitNo                   := #UnitNo,
           SpIRec                   := DB2041.LABOR_FREIG_T4,
           SpIBit                   := I    258.3);

NETWORK
TITLE =messages

      NOP   0;
// msg001 Msg 001 Message 01
      CALL FC    16 (
           UnitNo                   := #UnitNo,
           MsgRec                   := DB2047.msg001,
           MsgBit                   := DB2047.DBX   82.7);

// msg002 Msg 002 Message 02
      CALL FC    16 (
           UnitNo                   := #UnitNo,
           MsgRec                   := DB2047.msg002,
           MsgBit                   := DB2047.DBX  142.7);

NETWORK
TITLE =unit supply

      UC    FB [#UnitFB];

NETWORK
TITLE =T4_A10
// Act 005
// Box           : Ventilinsel 2
// Input address : I316.5
// Output address: Q316.5
      CALL FC    70 (
           UnitNo                   := #UnitNo,
           ActRec                   := DB2040.T4_A10,
           Typ                      := 1,
           FBa                      := #xTmp,
           FBa2                     := I    316.5,
           Out                      := Q    316.5);

NETWORK
TITLE =T4_A9
// Act 006
// Box           : Ventilinsel 2
// Input address : I318.5
// Output address: Q318.5
      CALL FC    70 (
           UnitNo                   := #UnitNo,
           ActRec                   := DB2040.T4_A9,
           Typ                      := 1,
           FBa                      := #xTmp,
           FBa2                     := I    318.5,
           Out                      := Q    318.5);

NETWORK
TITLE =T4_A12
// Act 007
// Box           : Ventilinsel 2
// Input address : I320.5
// Output address: Q320.5
      CALL FC    70 (
           UnitNo                   := #UnitNo,
           ActRec                   := DB2040.T4_A12,
           Typ                      := 1,
           FBa                      := #xTmp,
           FBa2                     := I    320.5,
           Out                      := Q    320.5);

NETWORK
TITLE =T4_A7
// Act 008
// Box           : Ventilinsel 2
// Input address : I322.5
// Output address: Q322.5
      CALL FC    70 (
           UnitNo                   := #UnitNo,
           ActRec                   := DB2040.T4_A7,
           Typ                      := 1,
           FBa                      := #xTmp,
           FBa2                     := I    322.5,
           Out                      := Q    322.5);

NETWORK
TITLE =T4_A8
// Act 009
// Box           : Ventilinsel 3
// Input address : I324.5
// Output address: Q324.5
      CALL FC    70 (
           UnitNo                   := #UnitNo,
           ActRec                   := DB2040.T4_A8,
           Typ                      := 1,
           FBa                      := #xTmp,
           FBa2                     := I    324.5,
           Out                      := Q    324.5);

NETWORK
TITLE =T4_A5
// Act 010
// Box           : Ventilinsel 3
// Input address : I326.5
// Output address: Q326.5
      CALL FC    70 (
           UnitNo                   := #UnitNo,
           ActRec                   := DB2040.T4_A5,
           Typ                      := 1,
           FBa                      := #xTmp,
           FBa2                     := I    326.5,
           Out                      := Q    326.5);

NETWORK
TITLE =T4_A11
// Act 011
// Box           : Ventilinsel 3
// Input address : I328.5
// Output address: Q328.5
      CALL FC    70 (
           UnitNo                   := #UnitNo,
           ActRec                   := DB2040.T4_A11,
           Typ                      := 1,
           FBa                      := #xTmp,
           FBa2                     := I    328.5,
           Out                      := Q    328.5);

NETWORK
TITLE =T4_A14
// Act 012
// Box           : Ventilinsel 4
// Input address : I330.5
// Output address: Q330.5
      CALL FC    70 (
           UnitNo                   := #UnitNo,
           ActRec                   := DB2040.T4_A14,
           Typ                      := 1,
           FBa                      := #xTmp,
           FBa2                     := I    330.5,
           Out                      := Q    330.5);

NETWORK
TITLE =T4_A15
// Act 013
// Box           : Ventilinsel 4
// Input address : I332.5
// Output address: Q332.5
      CALL FC    70 (
           UnitNo                   := #UnitNo,
           ActRec                   := DB2040.T4_A15,
           Typ                      := 0,
           FBa                      := #xTmp,
           FBa2                     := I    332.5,
           Out                      := Q    332.5);

NETWORK
TITLE =T4_RR1
// Act 014
// Box           : Ventilinsel 4
// Input address : I334.5
// Output address: Q334.5
      CALL FC    70 (
           UnitNo                   := #UnitNo,
           ActRec                   := DB2040.T4_RR1,
           Typ                      := 1,
           FBa                      := #xTmp,
           FBa2                     := I    334.5,
           Out                      := Q    334.5);

NETWORK
TITLE =RV1_T4  RV1_T4 Ventil CIP Vorlauf Tank 4
// Act 015
// Box           : VS1-BB
// Input address : I299.7
// Output address: Q299.7
      CALL FC    70 (
           UnitNo                   := #UnitNo,
           ActRec                   := DB2040.RV1_T4,
           Typ                      := 1,
           FBa                      := #xTmp,
           FBa2                     := I    299.7,
           Out                      := Q    299.7);

NETWORK
TITLE =B6F_T4  B6F_T4
// Act 016
// Box           : VS1-BB
// Input address : I300.3
// Output address: Q300.3
      CALL FC    70 (
           UnitNo                   := #UnitNo,
           ActRec                   := DB2040.B6F_T4,
           Typ                      := 1,
           FBa                      := #xTmp,
           FBa2                     := I    300.3,
           Out                      := Q    300.3);

NETWORK
TITLE =H6F_T4  H6F_T4
// Act 017
// Box           : VS1-BB
// Input address : I300.2
// Output address: Q300.2
      CALL FC    70 (
           UnitNo                   := #UnitNo,
           ActRec                   := DB2040.H6F_T4,
           Typ                      := 1,
           FBa                      := #xTmp,
           FBa2                     := I    300.2,
           Out                      := Q    300.2);

NETWORK
TITLE =J6F_T4  J6F_T4
// Act 018
// Box           : VS1-BB
// Input address : I300.4
// Output address: Q300.4
      CALL FC    70 (
           UnitNo                   := #UnitNo,
           ActRec                   := DB2040.J6F_T4,
           Typ                      := 1,
           FBa                      := #xTmp,
           FBa2                     := I    300.4,
           Out                      := Q    300.4);

NETWORK
TITLE =L6F_T4  L6F_T4
// Act 019
// Box           : VS1-BB
// Input address : I300.5
// Output address: Q300.5
      CALL FC    70 (
           UnitNo                   := #UnitNo,
           ActRec                   := DB2040.L6F_T4,
           Typ                      := 1,
           FBa                      := #xTmp,
           FBa2                     := I    300.5,
           Out                      := Q    300.5);

NETWORK
TITLE =D6_T4  D6_T4
// Act 020
// Box           : VS1-BB
// Input address : I300.7
// Output address: Q300.7
      CALL FC    70 (
           UnitNo                   := #UnitNo,
           ActRec                   := DB2040.D6_T4,
           Typ                      := 1,
           FBa                      := #xTmp,
           FBa2                     := I    300.7,
           Out                      := Q    300.7);

NETWORK
TITLE =B6_T4  B6_T4
// Act 021
// Box           : VS1-BB
// Input address : I300.6
// Output address: Q300.6
      CALL FC    70 (
           UnitNo                   := #UnitNo,
           ActRec                   := DB2040.B6_T4,
           Typ                      := 1,
           FBa                      := #xTmp,
           FBa2                     := I    300.6,
           Out                      := Q    300.6);

NETWORK
TITLE =A_T4  A_T4
// Act 022
// Box           : VS1-BB
// Input address : I300.0
// Output address: Q300.0
      CALL FC    70 (
           UnitNo                   := #UnitNo,
           ActRec                   := DB2040.A_T4,
           Typ                      := 1,
           FBa                      := #xTmp,
           FBa2                     := I    300.0,
           Out                      := Q    300.0);

NETWORK
TITLE =B_T4  B_T4
// Act 023
// Box           : VS1-BB
// Input address : I300.1
// Output address: Q300.1
      CALL FC    70 (
           UnitNo                   := #UnitNo,
           ActRec                   := DB2040.B_T4,
           Typ                      := 1,
           FBa                      := #xTmp,
           FBa2                     := I    300.1,
           Out                      := Q    300.1);

NETWORK
TITLE =CF_T4
// Act 024
// Box           : Ventilinsel 1
// Input address : I16.4
// Output address: Q16.4
      CALL FC    70 (
           UnitNo                   := #UnitNo,
           ActRec                   := DB2040.CF_T4,
           Typ                      := 1,
           FBa                      := #xTmp,
           FBa2                     := I     16.4,
           Out                      := Q     16.4);

NETWORK
TITLE =VR_T4  VR_T4
// Act 029
// Box           : VS1-BB
// Output address: Q301.0
      CALL FC    70 (
           UnitNo                   := #UnitNo,
           ActRec                   := DB2040.VR_T4,
           Typ                      := 0,
           FBa                      := #xTmp,
           FBa2                     := #xTmp,
           Out                      := Q    301.0);

NETWORK
TITLE =ML_LABORFREIGABE_T4
// Act 031
// Box           : LT-CIP
// Output address: Q258.3
      CALL FC    70 (
           UnitNo                   := #UnitNo,
           ActRec                   := DB2040.ML_LABORFREIGABE_T4,
           Typ                      := 0,
           FBa                      := #xTmp,
           FBa2                     := #xTmp,
           Out                      := Q    258.3);

END_FUNCTION_BLOCK

FUNCTION_BLOCK FB 1041
TITLE =U004: Water Tank 4
FAMILY : BOTEC_F1
NAME : UniE
VERSION : 1.2


VAR_TEMP
  CIP : BOOL ;	//CIP active
  UNIM : BOOL ;	//Unit Not In Maintenance
  GenRel : BOOL ;	//general OK (emergency and maintenance OK)
  EStopOK : BOOL ;	//emergency OK
  UnitNo : INT ;	//unit number
  xTmp : BOOL ;	//Temporary Bool
  iTmp : INT ;	//Temporary INT
  rTmp : REAL ;	//Temporary REAL
  dTmp : DINT ;	//Temporary DINT (free for general use)
  RetValInt : INT ;	//return value
END_VAR
BEGIN
NETWORK
TITLE =General

      SET   ;
// Simulation ---------------------------------------------------------------
      A     DB1041.DBX 1357.7;
      CC    FB  1049; // "WT04Sim"
      A     DB1041.DBX   17.3;
      =     DB1041.DBX 1357.7; //Help bit for simulation

// get unit number ----------------------------------------------------------
      L     DB1040.DBW    0;
      T     #UnitNo;

// communication ------------------------------------------------------------
      UC    FB  1045; // WT04Com

NETWORK
TITLE =Sequence organisation

      CLR   ;
      =     M    122.2;

// CIP Counter
      CALL FC    29 (
           UnitNo                   := #UnitNo,
           Value                    := DB1045.DBD   54,
           Enable                   := TRUE,
           Down                     := FALSE,
           OriginDetect             := 0.000000e+000,
           MaxDiffPS                := 1.000000e+000,
           SFMRec                   := DB1041.Seq.SFM[15],
           ValueOld                 := DB1041.DBD 1418);

// sequencer ----------------------------------------------------------------
      A     DB1043.DBX   43.1;
      S     DB1043.DBX   97.3;

      CALL FC    40 (
           UnitNo                   := #UnitNo);

END_FUNCTION_BLOCK

FUNCTION_BLOCK FB 1050
TITLE =U005: Wassertank 05
FAMILY : BOTEC_F1
NAME : U005A
VERSION : 2.1


VAR_TEMP
  EStopOK : BOOL ;	//auxiliary flag
  CIP : BOOL ;	//CIP Program Selected
  xTmp : BOOL ;	//Temporary Bool(free for general use)
  DummyBool : BOOL ;	//Temporary Bool(free for general use)
  UnitNo : INT ;	//unit number
  UnitFB : INT ;	//unit expansion FB number
  rTmp : REAL ;	//Temporary REAL (free for general use)
  iTmp : INT ;	//Temporary INT (free for general use)
  DummyInt : INT ;	//Temporary INT (free for general use)
  dTmp : DINT ;	//Temporary DINT (free for general use)
END_VAR
BEGIN
NETWORK
TITLE =general

      CLR   ;
      =     #xTmp;
      =     #EStopOK;

      L     DB1050.DBW    0;
      T     #UnitNo;
      L     DB1050.DBW    2;
      T     #UnitFB;

NETWORK
TITLE =analog inputs

      NOP   0;
// LI_T5 AnI 001 Inhalt Tank 5
      CALL FC    24 (
           UnitNo                   := #UnitNo,
           AnIRec                   := DB2053.LI_T5,
           ValPer                   := DB302.DBW   72);

NETWORK
TITLE =Universal value

      NOP   0;
// unv001 UnV 001 Process Status
      CALL FC    27 (
           UnitNo                   := #UnitNo,
           UnVRec                   := DB2055.unv001,
           ValExt                   := DB2055.DBD  234);

// unv002 UnV 002 Universal Value 02
      CALL FC    27 (
           UnitNo                   := #UnitNo,
           UnVRec                   := DB2055.unv002,
           ValExt                   := DB2055.DBD  362);

// unv003 UnV 003 Universal Value 03
      CALL FC    27 (
           UnitNo                   := #UnitNo,
           UnVRec                   := DB2055.unv003,
           ValExt                   := DB2055.DBD  490);

NETWORK
TITLE =special inputs

      NOP   0;
// LS_LLL_T5 SpI 001
      CALL FC    14 (
           UnitNo                   := #UnitNo,
           SpIRec                   := DB2051.LS_LLL_T5,
           SpIBit                   := I     67.7);

// LS_HL_T5 SpI 002
      CALL FC    14 (
           UnitNo                   := #UnitNo,
           SpIRec                   := DB2051.LS_HL_T5,
           SpIBit                   := I     67.5);

// LS_LL_T5 SpI 005
      CALL FC    14 (
           UnitNo                   := #UnitNo,
           SpIRec                   := DB2051.LS_LL_T5,
           SpIBit                   := I     67.6);

// T5_K4 SpI 006 RM Handklappe
//      CALL  "SI1"
//       UnitNo:=#UnitNo
//       SpIRec:="U005SpID".T5_K4
//       SpIBit:="T5_K4"

// RM_NI_T5_K2 SpI 008
      CALL FC    14 (
           UnitNo                   := #UnitNo,
           SpIRec                   := DB2051.RM_NI_T5_K2,
           SpIBit                   := I     61.0);

// RM_NI_T5_K3 SpI 010
      CALL FC    14 (
           UnitNo                   := #UnitNo,
           SpIRec                   := DB2051.RM_NI_T5_K3,
           SpIBit                   := I     69.2);

// LABOR_FREIG_T5 SpI 011 SCHLUESSELSCHALTER LABOR
      CALL FC    14 (
           UnitNo                   := #UnitNo,
           SpIRec                   := DB2051.LABOR_FREIG_T5,
           SpIBit                   := I    258.4);

NETWORK
TITLE =messages

      NOP   0;
// msg001 Msg 001 Message 01
      CALL FC    16 (
           UnitNo                   := #UnitNo,
           MsgRec                   := DB2057.msg001,
           MsgBit                   := DB2057.DBX   82.7);

// msg002 Msg 002 Message 02
      CALL FC    16 (
           UnitNo                   := #UnitNo,
           MsgRec                   := DB2057.msg002,
           MsgBit                   := DB2057.DBX  142.7);

NETWORK
TITLE =unit supply

      UC    FB [#UnitFB];

NETWORK
TITLE =T5_BH
// Act 002
// Box           : Ventilinsel 5
// Input address : I339.0
// Output address: Q339.0
      CALL FC    70 (
           UnitNo                   := #UnitNo,
           ActRec                   := DB2050.T5_BH,
           Typ                      := 1,
           FBa                      := #xTmp,
           FBa2                     := I    339.0,
           Out                      := Q    339.0);

NETWORK
TITLE =T5_KEG
// Act 003
// Box           : Ventilinsel 5
// Input address : I339.3
// Output address: Q339.3
      CALL FC    70 (
           UnitNo                   := #UnitNo,
           ActRec                   := DB2050.T5_KEG,
           Typ                      := 1,
           FBa                      := #xTmp,
           FBa2                     := I    339.3,
           Out                      := Q    339.3);

NETWORK
TITLE =T5_SK
// Act 004
// Box           : Ventilinsel 5
// Input address : I338.2
// Output address: Q338.2
      CALL FC    70 (
           UnitNo                   := #UnitNo,
           ActRec                   := DB2050.T5_SK,
           Typ                      := 1,
           FBa                      := #xTmp,
           FBa2                     := I    338.2,
           Out                      := Q    338.2);

NETWORK
TITLE =T5_A10
// Act 005
// Box           : Ventilinsel 2
// Input address : I316.4
// Output address: Q316.4
      CALL FC    70 (
           UnitNo                   := #UnitNo,
           ActRec                   := DB2050.T5_A10,
           Typ                      := 1,
           FBa                      := #xTmp,
           FBa2                     := I    316.4,
           Out                      := Q    316.4);

NETWORK
TITLE =T5_A9
// Act 006
// Box           : Ventilinsel 2
// Input address : I318.4
// Output address: Q318.4
      CALL FC    70 (
           UnitNo                   := #UnitNo,
           ActRec                   := DB2050.T5_A9,
           Typ                      := 1,
           FBa                      := #xTmp,
           FBa2                     := I    318.4,
           Out                      := Q    318.4);

NETWORK
TITLE =T5_A12
// Act 007
// Box           : Ventilinsel 2
// Input address : I320.4
// Output address: Q320.4
      CALL FC    70 (
           UnitNo                   := #UnitNo,
           ActRec                   := DB2050.T5_A12,
           Typ                      := 1,
           FBa                      := #xTmp,
           FBa2                     := I    320.4,
           Out                      := Q    320.4);

NETWORK
TITLE =T5_A7
// Act 008
// Box           : Ventilinsel 2
// Input address : I322.4
// Output address: Q322.4
      CALL FC    70 (
           UnitNo                   := #UnitNo,
           ActRec                   := DB2050.T5_A7,
           Typ                      := 1,
           FBa                      := #xTmp,
           FBa2                     := I    322.4,
           Out                      := Q    322.4);

NETWORK
TITLE =T5_A8
// Act 009
// Box           : Ventilinsel 3
// Input address : I324.4
// Output address: Q324.4
      CALL FC    70 (
           UnitNo                   := #UnitNo,
           ActRec                   := DB2050.T5_A8,
           Typ                      := 1,
           FBa                      := #xTmp,
           FBa2                     := I    324.4,
           Out                      := Q    324.4);

NETWORK
TITLE =T5_A5
// Act 010
// Box           : Ventilinsel 3
// Input address : I326.4
// Output address: Q326.4
      CALL FC    70 (
           UnitNo                   := #UnitNo,
           ActRec                   := DB2050.T5_A5,
           Typ                      := 1,
           FBa                      := #xTmp,
           FBa2                     := I    326.4,
           Out                      := Q    326.4);

NETWORK
TITLE =T5_A11
// Act 011
// Box           : Ventilinsel 3
// Input address : I328.4
// Output address: Q328.4
      CALL FC    70 (
           UnitNo                   := #UnitNo,
           ActRec                   := DB2050.T5_A11,
           Typ                      := 1,
           FBa                      := #xTmp,
           FBa2                     := I    328.4,
           Out                      := Q    328.4);

NETWORK
TITLE =T5_A14
// Act 012
// Box           : Ventilinsel 4
// Input address : I330.4
// Output address: Q330.4
      CALL FC    70 (
           UnitNo                   := #UnitNo,
           ActRec                   := DB2050.T5_A14,
           Typ                      := 1,
           FBa                      := #xTmp,
           FBa2                     := I    330.4,
           Out                      := Q    330.4);

NETWORK
TITLE =T5_A15
// Act 013
// Box           : Ventilinsel 4
// Input address : I332.4
// Output address: Q332.4
      CALL FC    70 (
           UnitNo                   := #UnitNo,
           ActRec                   := DB2050.T5_A15,
           Typ                      := 0,
           FBa                      := #xTmp,
           FBa2                     := I    332.4,
           Out                      := Q    332.4);

NETWORK
TITLE =T5_RR1
// Act 014
// Box           : Ventilinsel 4
// Input address : I334.4
// Output address: Q334.4
      CALL FC    70 (
           UnitNo                   := #UnitNo,
           ActRec                   := DB2050.T5_RR1,
           Typ                      := 1,
           FBa                      := #xTmp,
           FBa2                     := I    334.4,
           Out                      := Q    334.4);

NETWORK
TITLE =RV1_T5  RV1_T5 Ventil CIP Vorlauf Tank 5
// Act 015
// Box           : VS1-BB
// Input address : I301.1
// Output address: Q301.1
      CALL FC    70 (
           UnitNo                   := #UnitNo,
           ActRec                   := DB2050.RV1_T5,
           Typ                      := 1,
           FBa                      := #xTmp,
           FBa2                     := I    301.1,
           Out                      := Q    301.1);

NETWORK
TITLE =B6F_T5  B6F_T5
// Act 016
// Box           : VS1-BB
// Input address : I301.5
// Output address: Q301.5
      CALL FC    70 (
           UnitNo                   := #UnitNo,
           ActRec                   := DB2050.B6F_T5,
           Typ                      := 1,
           FBa                      := #xTmp,
           FBa2                     := I    301.5,
           Out                      := Q    301.5);

NETWORK
TITLE =H6F_T5  H6F_T5
// Act 017
// Box           : VS1-BB
// Input address : I301.4
// Output address: Q301.4
      CALL FC    70 (
           UnitNo                   := #UnitNo,
           ActRec                   := DB2050.H6F_T5,
           Typ                      := 1,
           FBa                      := #xTmp,
           FBa2                     := I    301.4,
           Out                      := Q    301.4);

NETWORK
TITLE =J6F_T5  J6F_T5
// Act 018
// Box           : VS1-BB
// Input address : I301.6
// Output address: Q301.6
      CALL FC    70 (
           UnitNo                   := #UnitNo,
           ActRec                   := DB2050.J6F_T5,
           Typ                      := 1,
           FBa                      := #xTmp,
           FBa2                     := I    301.6,
           Out                      := Q    301.6);

NETWORK
TITLE =L6F_T5  L6F_T5
// Act 019
// Box           : VS1-BB
// Input address : I301.7
// Output address: Q301.7
      CALL FC    70 (
           UnitNo                   := #UnitNo,
           ActRec                   := DB2050.L6F_T5,
           Typ                      := 1,
           FBa                      := #xTmp,
           FBa2                     := I    301.7,
           Out                      := Q    301.7);

NETWORK
TITLE =D6_T5  D6_T5
// Act 020
// Box           : VS1-BB
// Input address : I302.1
// Output address: Q302.1
      CALL FC    70 (
           UnitNo                   := #UnitNo,
           ActRec                   := DB2050.D6_T5,
           Typ                      := 1,
           FBa                      := #xTmp,
           FBa2                     := I    302.1,
           Out                      := Q    302.1);

NETWORK
TITLE =B6_T5  B6_T5
// Act 021
// Box           : VS1-BB
// Input address : I302.0
// Output address: Q302.0
      CALL FC    70 (
           UnitNo                   := #UnitNo,
           ActRec                   := DB2050.B6_T5,
           Typ                      := 1,
           FBa                      := #xTmp,
           FBa2                     := I    302.0,
           Out                      := Q    302.0);

NETWORK
TITLE =A_T5  A_T5
// Act 022
// Box           : VS1-BB
// Input address : I301.2
// Output address: Q301.2
      CALL FC    70 (
           UnitNo                   := #UnitNo,
           ActRec                   := DB2050.A_T5,
           Typ                      := 1,
           FBa                      := #xTmp,
           FBa2                     := I    301.2,
           Out                      := Q    301.2);

NETWORK
TITLE =B_T5  B_T5
// Act 023
// Box           : VS1-BB
// Input address : I301.3
// Output address: Q301.3
      CALL FC    70 (
           UnitNo                   := #UnitNo,
           ActRec                   := DB2050.B_T5,
           Typ                      := 1,
           FBa                      := #xTmp,
           FBa2                     := I    301.3,
           Out                      := Q    301.3);

NETWORK
TITLE =CF_T5
// Act 024
// Box           : Ventilinsel 1
// Input address : I16.6
// Output address: Q16.6
      CALL FC    70 (
           UnitNo                   := #UnitNo,
           ActRec                   := DB2050.CF_T5,
           Typ                      := 1,
           FBa                      := #xTmp,
           FBa2                     := I     16.6,
           Out                      := Q     16.6);

NETWORK
TITLE =RW5_T5  RW5_T5
// Act 026
// Box           : VS1-BB
// Input address : I302.2
// Output address: Q302.2
      CALL FC    70 (
           UnitNo                   := #UnitNo,
           ActRec                   := DB2050.RW5_T5,
           Typ                      := 1,
           FBa                      := #xTmp,
           FBa2                     := I    302.2,
           Out                      := Q    302.2);

NETWORK
TITLE =RW6_T5  RW6_T5
// Act 027
// Box           : VS1-BB
// Input address : I302.3
// Output address: Q302.3
      CALL FC    70 (
           UnitNo                   := #UnitNo,
           ActRec                   := DB2050.RW6_T5,
           Typ                      := 1,
           FBa                      := #xTmp,
           FBa2                     := I    302.3,
           Out                      := Q    302.3);

NETWORK
TITLE =VR_T5  VR_T5
// Act 029
// Box           : VS1-BB
// Output address: Q302.4
      CALL FC    70 (
           UnitNo                   := #UnitNo,
           ActRec                   := DB2050.VR_T5,
           Typ                      := 0,
           FBa                      := #xTmp,
           FBa2                     := #xTmp,
           Out                      := Q    302.4);

NETWORK
TITLE =ML_LABORFREIGABE_T5
// Act 031
// Box           : LT-CIP
// Output address: Q258.4
      CALL FC    70 (
           UnitNo                   := #UnitNo,
           ActRec                   := DB2050.ML_LABORFREIGABE_T5,
           Typ                      := 0,
           FBa                      := #xTmp,
           FBa2                     := #xTmp,
           Out                      := Q    258.4);

END_FUNCTION_BLOCK

FUNCTION_BLOCK FB 1051
TITLE =U005: Water Tank 5
FAMILY : BOTEC_F1
NAME : UniE
VERSION : 1.2


VAR_TEMP
  CIP : BOOL ;	//CIP active
  UNIM : BOOL ;	//Unit Not In Maintenance
  GenRel : BOOL ;	//general OK (emergency and maintenance OK)
  EStopOK : BOOL ;	//emergency OK
  UnitNo : INT ;	//unit number
  xTmp : BOOL ;	//Temporary Bool
  iTmp : INT ;	//Temporary INT
  rTmp : REAL ;	//Temporary REAL
  dTmp : DINT ;	//Temporary DINT (free for general use)
  RetValInt : INT ;	//return value
END_VAR
BEGIN
NETWORK
TITLE =General

      SET   ;
// Simulation ---------------------------------------------------------------
      A     DB1051.DBX 1357.7;
      CC    FB  1059; // "WT05Sim"
      A     DB1051.DBX   17.3;
      =     DB1051.DBX 1357.7; //Help bit for simulation

// get unit number ----------------------------------------------------------
      L     DB1050.DBW    0;
      T     #UnitNo;

// communication ------------------------------------------------------------
      UC    FB  1055; // WT05Com

NETWORK
TITLE =Sequence organisation

      CLR   ;
      =     M    122.2;

// CIP Counter
      CALL FC    29 (
           UnitNo                   := #UnitNo,
           Value                    := DB1055.DBD   54,
           Enable                   := TRUE,
           Down                     := FALSE,
           OriginDetect             := 0.000000e+000,
           MaxDiffPS                := 1.000000e+000,
           SFMRec                   := DB1051.Seq.SFM[15],
           ValueOld                 := DB1051.DBD 1418);

// sequencer ----------------------------------------------------------------
      A     DB1053.DBX   43.1;
      S     DB1053.DBX   97.3;

      CALL FC    40 (
           UnitNo                   := #UnitNo);

END_FUNCTION_BLOCK

FUNCTION_BLOCK FB 1060
TITLE =U006: Wassertank 06
FAMILY : BOTEC_F1
NAME : U006A
VERSION : 2.1


VAR_TEMP
  EStopOK : BOOL ;	//auxiliary flag
  CIP : BOOL ;	//CIP Program Selected
  xTmp : BOOL ;	//Temporary Bool(free for general use)
  DummyBool : BOOL ;	//Temporary Bool(free for general use)
  UnitNo : INT ;	//unit number
  UnitFB : INT ;	//unit expansion FB number
  rTmp : REAL ;	//Temporary REAL (free for general use)
  iTmp : INT ;	//Temporary INT (free for general use)
  DummyInt : INT ;	//Temporary INT (free for general use)
  dTmp : DINT ;	//Temporary DINT (free for general use)
END_VAR
BEGIN
NETWORK
TITLE =general

      CLR   ;
      =     #xTmp;
      =     #EStopOK;

      L     DB1060.DBW    0;
      T     #UnitNo;
      L     DB1060.DBW    2;
      T     #UnitFB;

NETWORK
TITLE =analog inputs

      NOP   0;
// LI_T6 AnI 001 Inhalt Tank 6
      CALL FC    24 (
           UnitNo                   := #UnitNo,
           AnIRec                   := DB2063.LI_T6,
           ValPer                   := DB302.DBW   74);

NETWORK
TITLE =Universal value

      NOP   0;
// unv001 UnV 001 Process Status
      CALL FC    27 (
           UnitNo                   := #UnitNo,
           UnVRec                   := DB2065.unv001,
           ValExt                   := DB2065.DBD  234);

// unv002 UnV 002 Universal Value 02
      CALL FC    27 (
           UnitNo                   := #UnitNo,
           UnVRec                   := DB2065.unv002,
           ValExt                   := DB2065.DBD  362);

// unv003 UnV 003 Universal Value 03
      CALL FC    27 (
           UnitNo                   := #UnitNo,
           UnVRec                   := DB2065.unv003,
           ValExt                   := DB2065.DBD  490);

NETWORK
TITLE =special inputs

      NOP   0;
// LS_LLL_T6 SpI 001
      CALL FC    14 (
           UnitNo                   := #UnitNo,
           SpIRec                   := DB2061.LS_LLL_T6,
           SpIBit                   := I     70.5);

// LS_HL_T6 SpI 002
      CALL FC    14 (
           UnitNo                   := #UnitNo,
           SpIRec                   := DB2061.LS_HL_T6,
           SpIBit                   := I     70.3);

// LS_LL_T6 SpI 005
      CALL FC    14 (
           UnitNo                   := #UnitNo,
           SpIRec                   := DB2061.LS_LL_T6,
           SpIBit                   := I     70.4);

// RM_NI_T6_K2 SpI 008
      CALL FC    14 (
           UnitNo                   := #UnitNo,
           SpIRec                   := DB2061.RM_NI_T6_K2,
           SpIBit                   := I     61.1);

// RM_NI_T6_K3 SpI 010
      CALL FC    14 (
           UnitNo                   := #UnitNo,
           SpIRec                   := DB2061.RM_NI_T6_K3,
           SpIBit                   := I     69.3);

// LABOR_FREIG_T6 SpI 011 SCHLUESSELSCHALTER LABOR
      CALL FC    14 (
           UnitNo                   := #UnitNo,
           SpIRec                   := DB2061.LABOR_FREIG_T6,
           SpIBit                   := I    258.5);

NETWORK
TITLE =messages

      NOP   0;
// msg001 Msg 001 Message 01
      CALL FC    16 (
           UnitNo                   := #UnitNo,
           MsgRec                   := DB2067.msg001,
           MsgBit                   := DB2067.DBX   82.7);

// msg002 Msg 002 Message 02
      CALL FC    16 (
           UnitNo                   := #UnitNo,
           MsgRec                   := DB2067.msg002,
           MsgBit                   := DB2067.DBX  142.7);

NETWORK
TITLE =unit supply

      UC    FB [#UnitFB];

NETWORK
TITLE =T6_FW
// Act 001
// Box           : Ventilinsel 5
// Input address : I338.4
// Output address: Q338.4
      CALL FC    70 (
           UnitNo                   := #UnitNo,
           ActRec                   := DB2060.T6_FW,
           Typ                      := 1,
           FBa                      := #xTmp,
           FBa2                     := I    338.4,
           Out                      := Q    338.4);

NETWORK
TITLE =T6_KEG
// Act 003
// Box           : Ventilinsel 5
// Input address : I339.2
// Output address: Q339.2
      CALL FC    70 (
           UnitNo                   := #UnitNo,
           ActRec                   := DB2060.T6_KEG,
           Typ                      := 1,
           FBa                      := #xTmp,
           FBa2                     := I    339.2,
           Out                      := Q    339.2);

NETWORK
TITLE =T6_SK
// Act 004
// Box           : Ventilinsel 5
// Input address : I338.1
// Output address: Q338.1
      CALL FC    70 (
           UnitNo                   := #UnitNo,
           ActRec                   := DB2060.T6_SK,
           Typ                      := 1,
           FBa                      := #xTmp,
           FBa2                     := I    338.1,
           Out                      := Q    338.1);

NETWORK
TITLE =T6_A10
// Act 005
// Box           : Ventilinsel 2
// Input address : I316.3
// Output address: Q316.3
      CALL FC    70 (
           UnitNo                   := #UnitNo,
           ActRec                   := DB2060.T6_A10,
           Typ                      := 1,
           FBa                      := #xTmp,
           FBa2                     := I    316.3,
           Out                      := Q    316.3);

NETWORK
TITLE =T6_A9
// Act 006
// Box           : Ventilinsel 2
// Input address : I318.3
// Output address: Q318.3
      CALL FC    70 (
           UnitNo                   := #UnitNo,
           ActRec                   := DB2060.T6_A9,
           Typ                      := 1,
           FBa                      := #xTmp,
           FBa2                     := I    318.3,
           Out                      := Q    318.3);

NETWORK
TITLE =T6_A12
// Act 007
// Box           : Ventilinsel 2
// Input address : I320.3
// Output address: Q320.3
      CALL FC    70 (
           UnitNo                   := #UnitNo,
           ActRec                   := DB2060.T6_A12,
           Typ                      := 1,
           FBa                      := #xTmp,
           FBa2                     := I    320.3,
           Out                      := Q    320.3);

NETWORK
TITLE =T6_A7
// Act 008
// Box           : Ventilinsel 2
// Input address : I322.3
// Output address: Q322.3
      CALL FC    70 (
           UnitNo                   := #UnitNo,
           ActRec                   := DB2060.T6_A7,
           Typ                      := 1,
           FBa                      := #xTmp,
           FBa2                     := I    322.3,
           Out                      := Q    322.3);

NETWORK
TITLE =T6_A8
// Act 009
// Box           : Ventilinsel 3
// Input address : I324.3
// Output address: Q324.3
      CALL FC    70 (
           UnitNo                   := #UnitNo,
           ActRec                   := DB2060.T6_A8,
           Typ                      := 1,
           FBa                      := #xTmp,
           FBa2                     := I    324.3,
           Out                      := Q    324.3);

NETWORK
TITLE =T6_A5
// Act 010
// Box           : Ventilinsel 3
// Input address : I326.3
// Output address: Q326.3
      CALL FC    70 (
           UnitNo                   := #UnitNo,
           ActRec                   := DB2060.T6_A5,
           Typ                      := 1,
           FBa                      := #xTmp,
           FBa2                     := I    326.3,
           Out                      := Q    326.3);

NETWORK
TITLE =T6_A11
// Act 011
// Box           : Ventilinsel 3
// Input address : I328.3
// Output address: Q328.3
      CALL FC    70 (
           UnitNo                   := #UnitNo,
           ActRec                   := DB2060.T6_A11,
           Typ                      := 1,
           FBa                      := #xTmp,
           FBa2                     := I    328.3,
           Out                      := Q    328.3);

NETWORK
TITLE =T6_A14
// Act 012
// Box           : Ventilinsel 4
// Input address : I330.3
// Output address: Q330.3
      CALL FC    70 (
           UnitNo                   := #UnitNo,
           ActRec                   := DB2060.T6_A14,
           Typ                      := 1,
           FBa                      := #xTmp,
           FBa2                     := I    330.3,
           Out                      := Q    330.3);

NETWORK
TITLE =T6_A15
// Act 013
// Box           : Ventilinsel 4
// Input address : I332.3
// Output address: Q332.3
      CALL FC    70 (
           UnitNo                   := #UnitNo,
           ActRec                   := DB2060.T6_A15,
           Typ                      := 0,
           FBa                      := #xTmp,
           FBa2                     := I    332.3,
           Out                      := Q    332.3);

NETWORK
TITLE =T6_RR1
// Act 014
// Box           : Ventilinsel 4
// Input address : I334.3
// Output address: Q334.3
      CALL FC    70 (
           UnitNo                   := #UnitNo,
           ActRec                   := DB2060.T6_RR1,
           Typ                      := 1,
           FBa                      := #xTmp,
           FBa2                     := I    334.3,
           Out                      := Q    334.3);

NETWORK
TITLE =RV1_T6  RV1_T3 Ventil CIP Vorlauf Tank 6
// Act 015
// Box           : VS1-BB
// Input address : I302.5
// Output address: Q302.5
      CALL FC    70 (
           UnitNo                   := #UnitNo,
           ActRec                   := DB2060.RV1_T6,
           Typ                      := 1,
           FBa                      := #xTmp,
           FBa2                     := I    302.5,
           Out                      := Q    302.5);

NETWORK
TITLE =B6F_T6  B6F_T6
// Act 016
// Box           : VS1-BB
// Input address : I303.1
// Output address: Q303.1
      CALL FC    70 (
           UnitNo                   := #UnitNo,
           ActRec                   := DB2060.B6F_T6,
           Typ                      := 1,
           FBa                      := #xTmp,
           FBa2                     := I    303.1,
           Out                      := Q    303.1);

NETWORK
TITLE =H6F_T6  H6F_T6
// Act 017
// Box           : VS1-BB
// Input address : I303.0
// Output address: Q303.0
      CALL FC    70 (
           UnitNo                   := #UnitNo,
           ActRec                   := DB2060.H6F_T6,
           Typ                      := 1,
           FBa                      := #xTmp,
           FBa2                     := I    303.0,
           Out                      := Q    303.0);

NETWORK
TITLE =J6F_T6  J6F_T6
// Act 018
// Box           : VS1-BB
// Input address : I303.2
// Output address: Q303.2
      CALL FC    70 (
           UnitNo                   := #UnitNo,
           ActRec                   := DB2060.J6F_T6,
           Typ                      := 1,
           FBa                      := #xTmp,
           FBa2                     := I    303.2,
           Out                      := Q    303.2);

NETWORK
TITLE =L6F_T6  L6F_T6
// Act 019
// Box           : VS1-BB
// Input address : I303.3
// Output address: Q303.3
      CALL FC    70 (
           UnitNo                   := #UnitNo,
           ActRec                   := DB2060.L6F_T6,
           Typ                      := 1,
           FBa                      := #xTmp,
           FBa2                     := I    303.3,
           Out                      := Q    303.3);

NETWORK
TITLE =D6_T6  D6_T6
// Act 020
// Box           : VS1-BB
// Input address : I303.5
// Output address: Q303.5
      CALL FC    70 (
           UnitNo                   := #UnitNo,
           ActRec                   := DB2060.D6_T6,
           Typ                      := 1,
           FBa                      := #xTmp,
           FBa2                     := I    303.5,
           Out                      := Q    303.5);

NETWORK
TITLE =B6_T6  B6_T6
// Act 021
// Box           : VS1-BB
// Input address : I303.4
// Output address: Q303.4
      CALL FC    70 (
           UnitNo                   := #UnitNo,
           ActRec                   := DB2060.B6_T6,
           Typ                      := 1,
           FBa                      := #xTmp,
           FBa2                     := I    303.4,
           Out                      := Q    303.4);

NETWORK
TITLE =A_T6  A_T6
// Act 022
// Box           : VS1-BB
// Input address : I302.6
// Output address: Q302.6
      CALL FC    70 (
           UnitNo                   := #UnitNo,
           ActRec                   := DB2060.A_T6,
           Typ                      := 1,
           FBa                      := #xTmp,
           FBa2                     := I    302.6,
           Out                      := Q    302.6);

NETWORK
TITLE =B_T6  B_T6
// Act 023
// Box           : VS1-BB
// Input address : I302.7
// Output address: Q302.7
      CALL FC    70 (
           UnitNo                   := #UnitNo,
           ActRec                   := DB2060.B_T6,
           Typ                      := 1,
           FBa                      := #xTmp,
           FBa2                     := I    302.7,
           Out                      := Q    302.7);

NETWORK
TITLE =CF_T6
// Act 024
// Box           : Ventilinsel 1
// Input address : I16.7
// Output address: Q16.7
      CALL FC    70 (
           UnitNo                   := #UnitNo,
           ActRec                   := DB2060.CF_T6,
           Typ                      := 1,
           FBa                      := #xTmp,
           FBa2                     := I     16.7,
           Out                      := Q     16.7);

NETWORK
TITLE =RW5_T6  RW5_T6
// Act 026
// Box           : VS1-BB
// Input address : I303.6
// Output address: Q303.6
      CALL FC    70 (
           UnitNo                   := #UnitNo,
           ActRec                   := DB2060.RW5_T6,
           Typ                      := 1,
           FBa                      := #xTmp,
           FBa2                     := I    303.6,
           Out                      := Q    303.6);

NETWORK
TITLE =RW6_T6  RW6_T6
// Act 027
// Box           : VS1-BB
// Input address : I303.7
// Output address: Q303.7
      CALL FC    70 (
           UnitNo                   := #UnitNo,
           ActRec                   := DB2060.RW6_T6,
           Typ                      := 1,
           FBa                      := #xTmp,
           FBa2                     := I    303.7,
           Out                      := Q    303.7);

NETWORK
TITLE =VR_T6  VR_T6
// Act 029
// Box           : VS2-BB
// Output address: Q304.0
      CALL FC    70 (
           UnitNo                   := #UnitNo,
           ActRec                   := DB2060.VR_T6,
           Typ                      := 0,
           FBa                      := #xTmp,
           FBa2                     := #xTmp,
           Out                      := Q    304.0);

